Fanuc KAREL source: V_CAM_CHECK.kl

PROGRAM T
%NOLOCKGROUP
VAR
 v0 : STRING[40]
 v1 : BOOLEAN
 v2 : INTEGER
BEGIN
 V_CAM_CHECK(v0, v1, v2)
END T
